// Mitsubishi GX Developer project: 101-Aug09_20121119   PLC: FX1N

PROGRAM MAIN
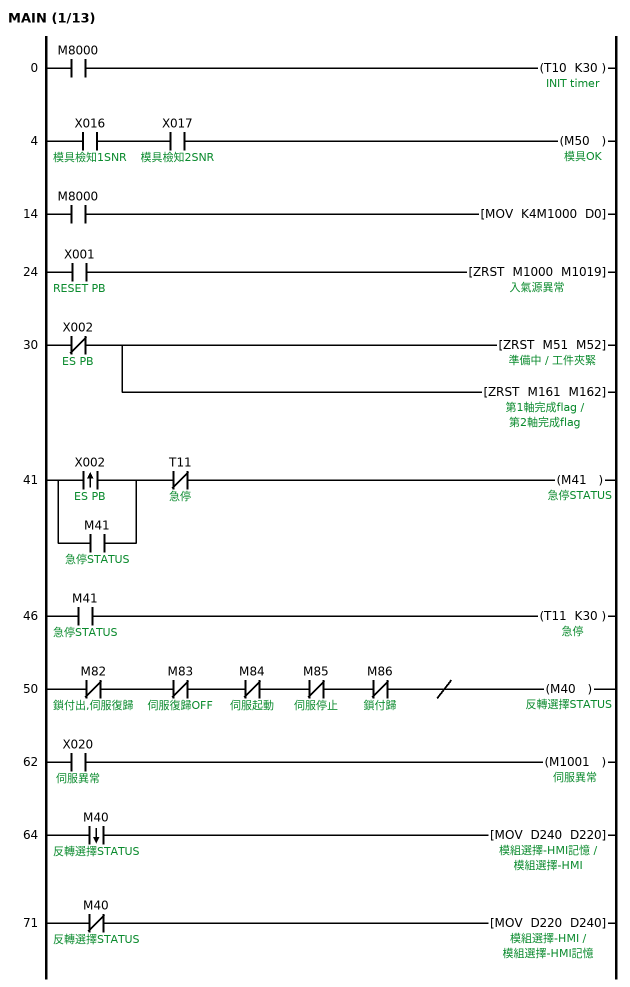
0     LD      M8000
      OUT     T10 K30  ; INIT timer
4     LD      X016  ; 模具檢知1SNR
      AND     X017  ; 模具檢知2SNR
      OUT     M50  ; 模具OK
14    LD      M8000
      MOV     K4M1000 D0  ; 入氣源異常
24    LD      X001  ; RESET PB
      ZRST    M1000 M1019
30    LDI     X002  ; ES PB
      ZRST    M51 M52  ; 準備中 / 工件夾緊
      ZRST    M161 M162  ; 第1軸完成flag / 第2軸完成flag
41    LDP     X002  ; ES PB
      OR      M41  ; 急停STATUS
      ANI     T11  ; 急停
      OUT     M41  ; 急停STATUS
46    LD      M41  ; 急停STATUS
      OUT     T11 K30  ; 急停
50    LDI     M82  ; 鎖付出,伺服復歸
      ANI     M83  ; 伺服復歸OFF
      ANI     M84  ; 伺服起動
      ANI     M85  ; 伺服停止
      ANI     M86  ; 鎖付歸
      INV
      OUT     M40  ; 反轉選擇STATUS
62    LD      X020  ; 伺服異常
      OUT     M1001  ; 伺服異常
64    LDF     M40  ; 反轉選擇STATUS
      MOV     D240 D220  ; 模組選擇-HMI記憶 / 模組選擇-HMI
71    LDI     M40  ; 反轉選擇STATUS
      MOV     D220 D240
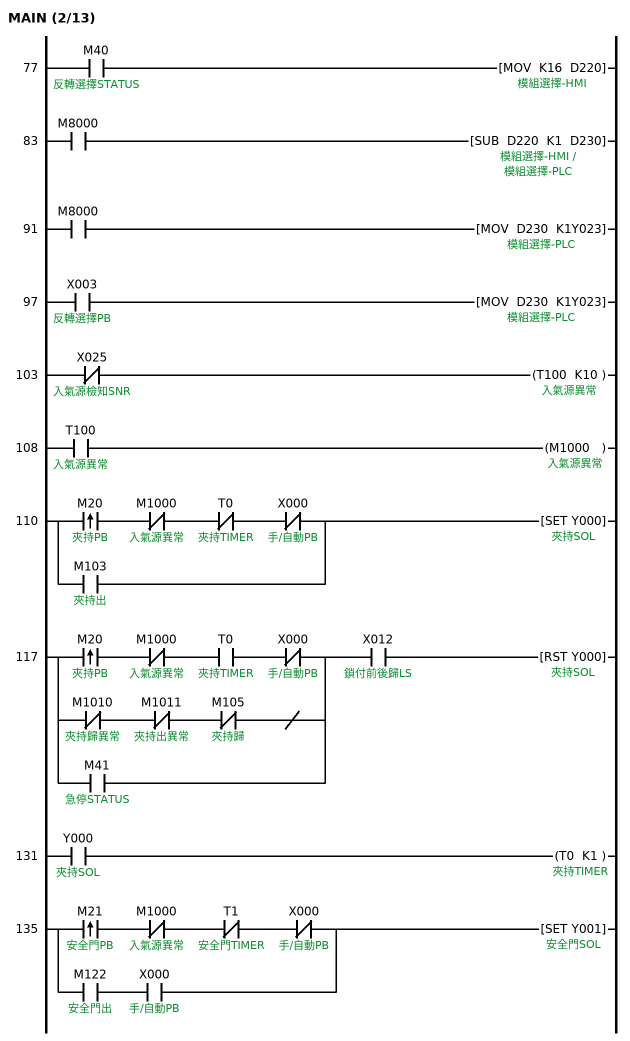
77    LD      M40  ; 反轉選擇STATUS
      MOV     K16 D220
83    LD      M8000
      SUB     D220 K1 D230  ; 模組選擇-PLC
91    LD      M8000
      MOV     D230 K1Y023  ; 工件選擇0
97    LD      X003  ; 反轉選擇PB
      MOV     D230 K1Y023
103   LDI     X025  ; 入氣源檢知SNR
      OUT     T100 K10  ; 入氣源異常
108   LD      T100  ; 入氣源異常
      OUT     M1000  ; 入氣源異常
110   LDP     M20  ; 夾持PB
      ANI     M1000  ; 入氣源異常
      ANI     T0  ; 夾持TIMER
      ANI     X000  ; 手/自動PB
      OR      M103  ; 夾持出
      SET     Y000  ; 夾持SOL
117   LDP     M20  ; 夾持PB
      ANI     M1000  ; 入氣源異常
      AND     T0  ; 夾持TIMER
      ANI     X000  ; 手/自動PB
      LDI     M1010  ; 夾持歸異常
      ANI     M1011  ; 夾持出異常
      ANI     M105  ; 夾持歸
      INV
      ORB
      OR      M41  ; 急停STATUS
      AND     X012  ; 鎖付前後歸LS
      RST     Y000  ; 夾持SOL
131   LD      Y000  ; 夾持SOL
      OUT     T0 K1  ; 夾持TIMER
135   LDP     M21  ; 安全門PB
      ANI     M1000  ; 入氣源異常
      ANI     T1  ; 安全門TIMER
      ANI     X000  ; 手/自動PB
      LD      M122  ; 安全門出
      AND     X000  ; 手/自動PB
      ORB
      SET     Y001  ; 安全門SOL
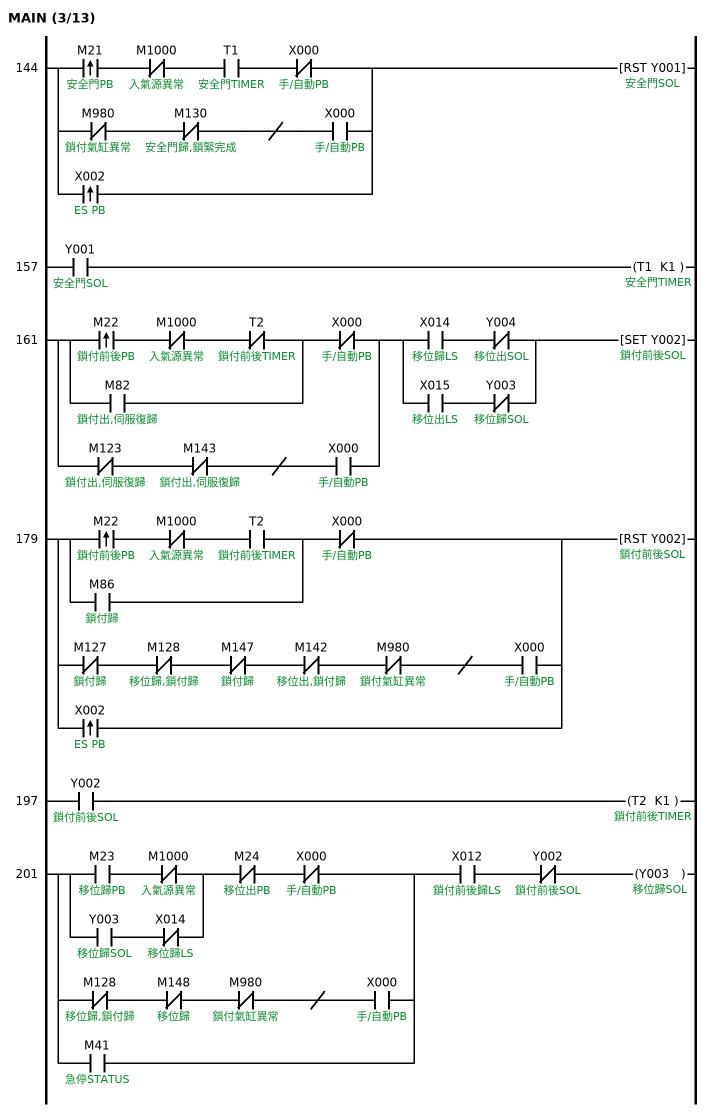
144   LDP     M21  ; 安全門PB
      ANI     M1000  ; 入氣源異常
      AND     T1  ; 安全門TIMER
      ANI     X000  ; 手/自動PB
      LDI     M980  ; 鎖付氣缸異常
      ANI     M130  ; 安全門歸,鎖緊完成
      INV
      AND     X000  ; 手/自動PB
      ORB
      ORP     X002  ; ES PB
      RST     Y001  ; 安全門SOL
157   LD      Y001  ; 安全門SOL
      OUT     T1 K1  ; 安全門TIMER
161   LDP     M22  ; 鎖付前後PB
      ANI     M1000  ; 入氣源異常
      ANI     T2  ; 鎖付前後TIMER
      OR      M82  ; 鎖付出,伺服復歸
      ANI     X000  ; 手/自動PB
      LDI     M123  ; 鎖付出,伺服復歸
      ANI     M143  ; 鎖付出,伺服復歸
      INV
      AND     X000  ; 手/自動PB
      ORB
      LD      X014  ; 移位歸LS
      ANI     Y004  ; 移位出SOL
      LD      X015  ; 移位出LS
      ANI     Y003  ; 移位歸SOL
      ORB
      ANB
      SET     Y002  ; 鎖付前後SOL
179   LDP     M22  ; 鎖付前後PB
      ANI     M1000  ; 入氣源異常
      AND     T2  ; 鎖付前後TIMER
      OR      M86  ; 鎖付歸
      ANI     X000  ; 手/自動PB
      LDI     M127  ; 鎖付歸
      ANI     M128  ; 移位歸,鎖付歸
      ANI     M147  ; 鎖付歸
      ANI     M142  ; 移位出,鎖付歸
      ANI     M980  ; 鎖付氣缸異常
      INV
      AND     X000  ; 手/自動PB
      ORB
      ORP     X002  ; ES PB
      RST     Y002  ; 鎖付前後SOL
197   LD      Y002  ; 鎖付前後SOL
      OUT     T2 K1  ; 鎖付前後TIMER
201   LD      M23  ; 移位歸PB
      ANI     M1000  ; 入氣源異常
      LD      Y003  ; 移位歸SOL
      ANI     X014  ; 移位歸LS
      ORB
      ANI     M24  ; 移位出PB
      ANI     X000  ; 手/自動PB
      LDI     M128  ; 移位歸,鎖付歸
      ANI     M148  ; 移位歸
      ANI     M980  ; 鎖付氣缸異常
      INV
      AND     X000  ; 手/自動PB
      ORB
      OR      M41  ; 急停STATUS
      AND     X012  ; 鎖付前後歸LS
      ANI     Y002  ; 鎖付前後SOL
      OUT     Y003  ; 移位歸SOL
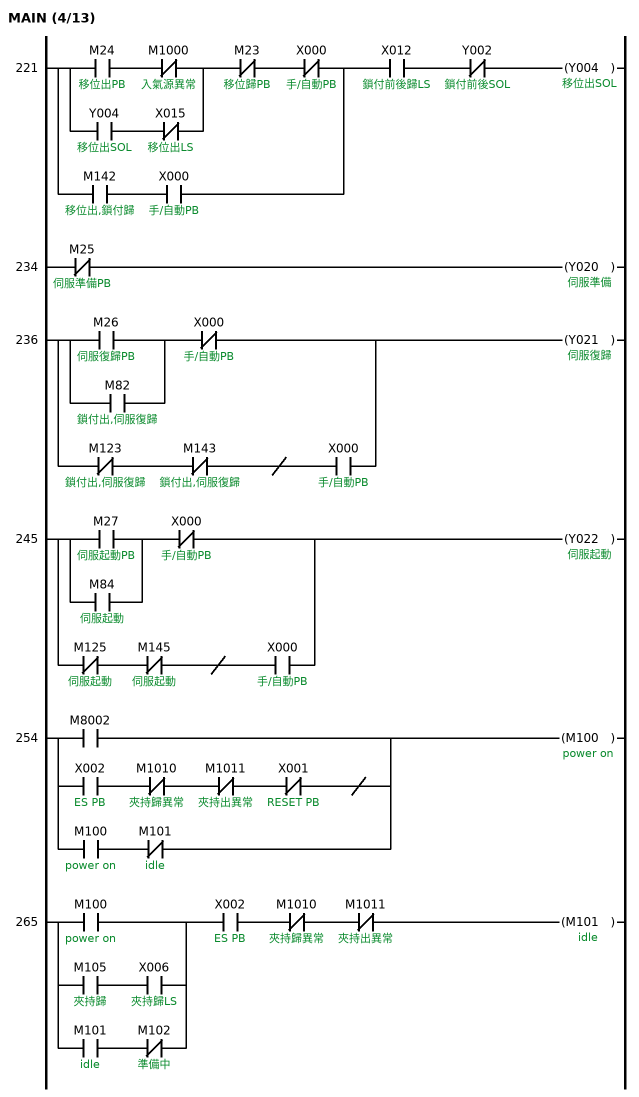
221   LD      M24  ; 移位出PB
      ANI     M1000  ; 入氣源異常
      LD      Y004  ; 移位出SOL
      ANI     X015  ; 移位出LS
      ORB
      ANI     M23  ; 移位歸PB
      ANI     X000  ; 手/自動PB
      LD      M142  ; 移位出,鎖付歸
      AND     X000  ; 手/自動PB
      ORB
      AND     X012  ; 鎖付前後歸LS
      ANI     Y002  ; 鎖付前後SOL
      OUT     Y004  ; 移位出SOL
234   LDI     M25  ; 伺服準備PB
      OUT     Y020  ; 伺服準備
236   LD      M26  ; 伺服復歸PB
      OR      M82  ; 鎖付出,伺服復歸
      ANI     X000  ; 手/自動PB
      LDI     M123  ; 鎖付出,伺服復歸
      ANI     M143  ; 鎖付出,伺服復歸
      INV
      AND     X000  ; 手/自動PB
      ORB
      OUT     Y021  ; 伺服復歸
245   LD      M27  ; 伺服起動PB
      OR      M84  ; 伺服起動
      ANI     X000  ; 手/自動PB
      LDI     M125  ; 伺服起動
      ANI     M145  ; 伺服起動
      INV
      AND     X000  ; 手/自動PB
      ORB
      OUT     Y022  ; 伺服起動
254   LD      M8002
      LD      X002  ; ES PB
      ANI     M1010  ; 夾持歸異常
      ANI     M1011  ; 夾持出異常
      ANI     X001  ; RESET PB
      INV
      ORB
      LD      M100  ; power on
      ANI     M101  ; idle
      ORB
      OUT     M100  ; power on
265   LD      M100  ; power on
      LD      M105  ; 夾持歸
      AND     X006  ; 夾持歸LS
      ORB
      LD      M101  ; idle
      ANI     M102  ; 準備中
      ORB
      AND     X002  ; ES PB
      ANI     M1010  ; 夾持歸異常
      ANI     M1011  ; 夾持出異常
      OUT     M101  ; idle
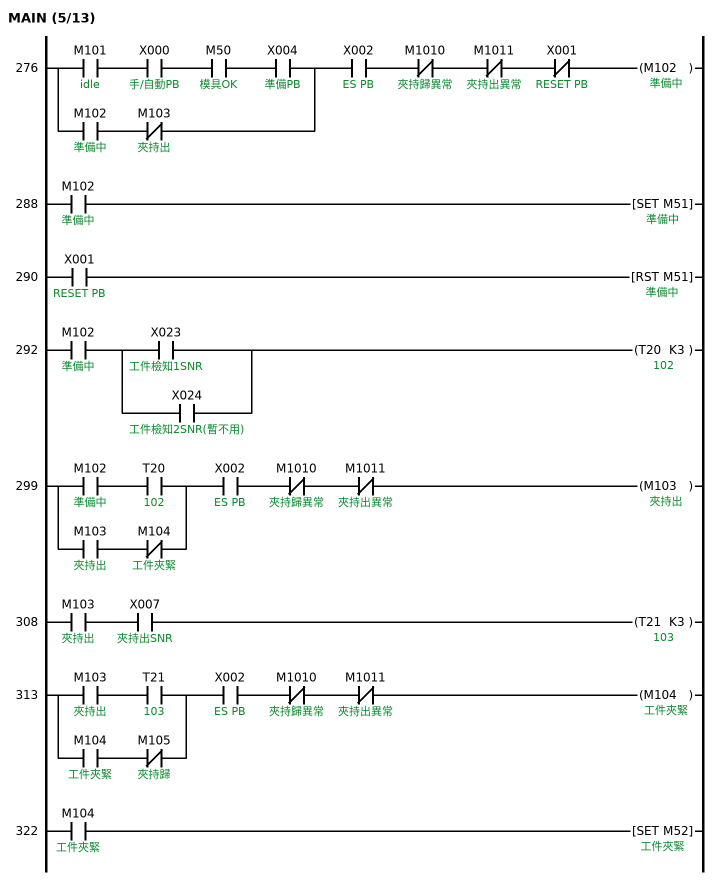
276   LD      M101  ; idle
      AND     X000  ; 手/自動PB
      AND     M50  ; 模具OK
      AND     X004  ; 準備PB
      LD      M102  ; 準備中
      ANI     M103  ; 夾持出
      ORB
      AND     X002  ; ES PB
      ANI     M1010  ; 夾持歸異常
      ANI     M1011  ; 夾持出異常
      ANI     X001  ; RESET PB
      OUT     M102  ; 準備中
288   LD      M102  ; 準備中
      SET     M51  ; 準備中
290   LD      X001  ; RESET PB
      RST     M51  ; 準備中
292   LD      M102  ; 準備中
      LD      X023  ; 工件檢知1SNR
      OR      X024  ; 工件檢知2SNR(暫不用)
      ANB
      OUT     T20 K3  ; 102
299   LD      M102  ; 準備中
      AND     T20  ; 102
      LD      M103  ; 夾持出
      ANI     M104  ; 工件夾緊
      ORB
      AND     X002  ; ES PB
      ANI     M1010  ; 夾持歸異常
      ANI     M1011  ; 夾持出異常
      OUT     M103  ; 夾持出
308   LD      M103  ; 夾持出
      AND     X007  ; 夾持出SNR
      OUT     T21 K3  ; 103
313   LD      M103  ; 夾持出
      AND     T21  ; 103
      LD      M104  ; 工件夾緊
      ANI     M105  ; 夾持歸
      ORB
      AND     X002  ; ES PB
      ANI     M1010  ; 夾持歸異常
      ANI     M1011  ; 夾持出異常
      OUT     M104  ; 工件夾緊
322   LD      M104  ; 工件夾緊
      SET     M52  ; 工件夾緊
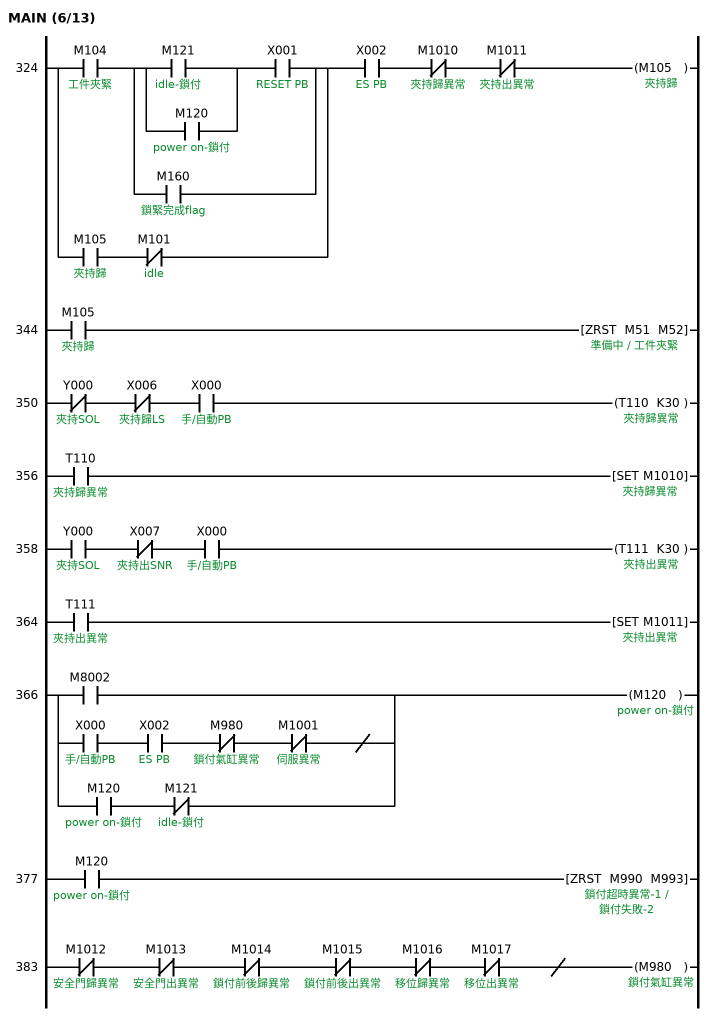
324   LD      M104  ; 工件夾緊
      LD      M121  ; idle-鎖付
      OR      M120  ; power on-鎖付
      AND     X001  ; RESET PB
      OR      M160  ; 鎖緊完成flag
      ANB
      LD      M105  ; 夾持歸
      ANI     M101  ; idle
      ORB
      AND     X002  ; ES PB
      ANI     M1010  ; 夾持歸異常
      ANI     M1011  ; 夾持出異常
      OUT     M105  ; 夾持歸
344   LD      M105  ; 夾持歸
      ZRST    M51 M52
350   LDI     Y000  ; 夾持SOL
      ANI     X006  ; 夾持歸LS
      AND     X000  ; 手/自動PB
      OUT     T110 K30  ; 夾持歸異常
356   LD      T110  ; 夾持歸異常
      SET     M1010  ; 夾持歸異常
358   LD      Y000  ; 夾持SOL
      ANI     X007  ; 夾持出SNR
      AND     X000  ; 手/自動PB
      OUT     T111 K30  ; 夾持出異常
364   LD      T111  ; 夾持出異常
      SET     M1011  ; 夾持出異常
366   LD      M8002
      LD      X000  ; 手/自動PB
      AND     X002  ; ES PB
      ANI     M980  ; 鎖付氣缸異常
      ANI     M1001  ; 伺服異常
      INV
      ORB
      LD      M120  ; power on-鎖付
      ANI     M121  ; idle-鎖付
      ORB
      OUT     M120  ; power on-鎖付
377   LD      M120  ; power on-鎖付
      ZRST    M990 M993  ; 鎖付超時異常-1 / 鎖付失敗-2
383   LDI     M1012  ; 安全門歸異常
      ANI     M1013  ; 安全門出異常
      ANI     M1014  ; 鎖付前後歸異常
      ANI     M1015  ; 鎖付前後出異常
      ANI     M1016  ; 移位歸異常
      ANI     M1017  ; 移位出異常
      INV
      OUT     M980  ; 鎖付氣缸異常
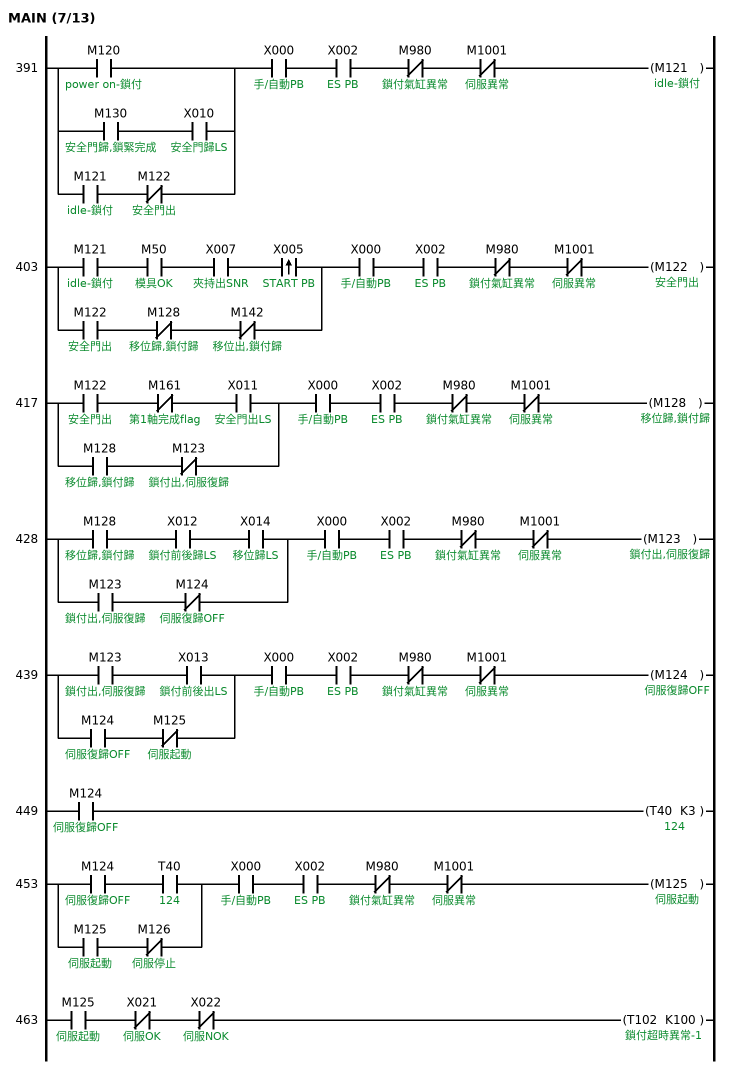
391   LD      M120  ; power on-鎖付
      LD      M130  ; 安全門歸,鎖緊完成
      AND     X010  ; 安全門歸LS
      ORB
      LD      M121  ; idle-鎖付
      ANI     M122  ; 安全門出
      ORB
      AND     X000  ; 手/自動PB
      AND     X002  ; ES PB
      ANI     M980  ; 鎖付氣缸異常
      ANI     M1001  ; 伺服異常
      OUT     M121  ; idle-鎖付
403   LD      M121  ; idle-鎖付
      AND     M50  ; 模具OK
      AND     X007  ; 夾持出SNR
      ANDP    X005  ; START PB
      LD      M122  ; 安全門出
      ANI     M128  ; 移位歸,鎖付歸
      ANI     M142  ; 移位出,鎖付歸
      ORB
      AND     X000  ; 手/自動PB
      AND     X002  ; ES PB
      ANI     M980  ; 鎖付氣缸異常
      ANI     M1001  ; 伺服異常
      OUT     M122  ; 安全門出
417   LD      M122  ; 安全門出
      ANI     M161  ; 第1軸完成flag
      AND     X011  ; 安全門出LS
      LD      M128  ; 移位歸,鎖付歸
      ANI     M123  ; 鎖付出,伺服復歸
      ORB
      AND     X000  ; 手/自動PB
      AND     X002  ; ES PB
      ANI     M980  ; 鎖付氣缸異常
      ANI     M1001  ; 伺服異常
      OUT     M128  ; 移位歸,鎖付歸
428   LD      M128  ; 移位歸,鎖付歸
      AND     X012  ; 鎖付前後歸LS
      AND     X014  ; 移位歸LS
      LD      M123  ; 鎖付出,伺服復歸
      ANI     M124  ; 伺服復歸OFF
      ORB
      AND     X000  ; 手/自動PB
      AND     X002  ; ES PB
      ANI     M980  ; 鎖付氣缸異常
      ANI     M1001  ; 伺服異常
      OUT     M123  ; 鎖付出,伺服復歸
439   LD      M123  ; 鎖付出,伺服復歸
      AND     X013  ; 鎖付前後出LS
      LD      M124  ; 伺服復歸OFF
      ANI     M125  ; 伺服起動
      ORB
      AND     X000  ; 手/自動PB
      AND     X002  ; ES PB
      ANI     M980  ; 鎖付氣缸異常
      ANI     M1001  ; 伺服異常
      OUT     M124  ; 伺服復歸OFF
449   LD      M124  ; 伺服復歸OFF
      OUT     T40 K3  ; 124
453   LD      M124  ; 伺服復歸OFF
      AND     T40  ; 124
      LD      M125  ; 伺服起動
      ANI     M126  ; 伺服停止
      ORB
      AND     X000  ; 手/自動PB
      AND     X002  ; ES PB
      ANI     M980  ; 鎖付氣缸異常
      ANI     M1001  ; 伺服異常
      OUT     M125  ; 伺服起動
463   LD      M125  ; 伺服起動
      ANI     X021  ; 伺服OK
      ANI     X022  ; 伺服NOK
      OUT     T102 K100  ; 鎖付超時異常-1
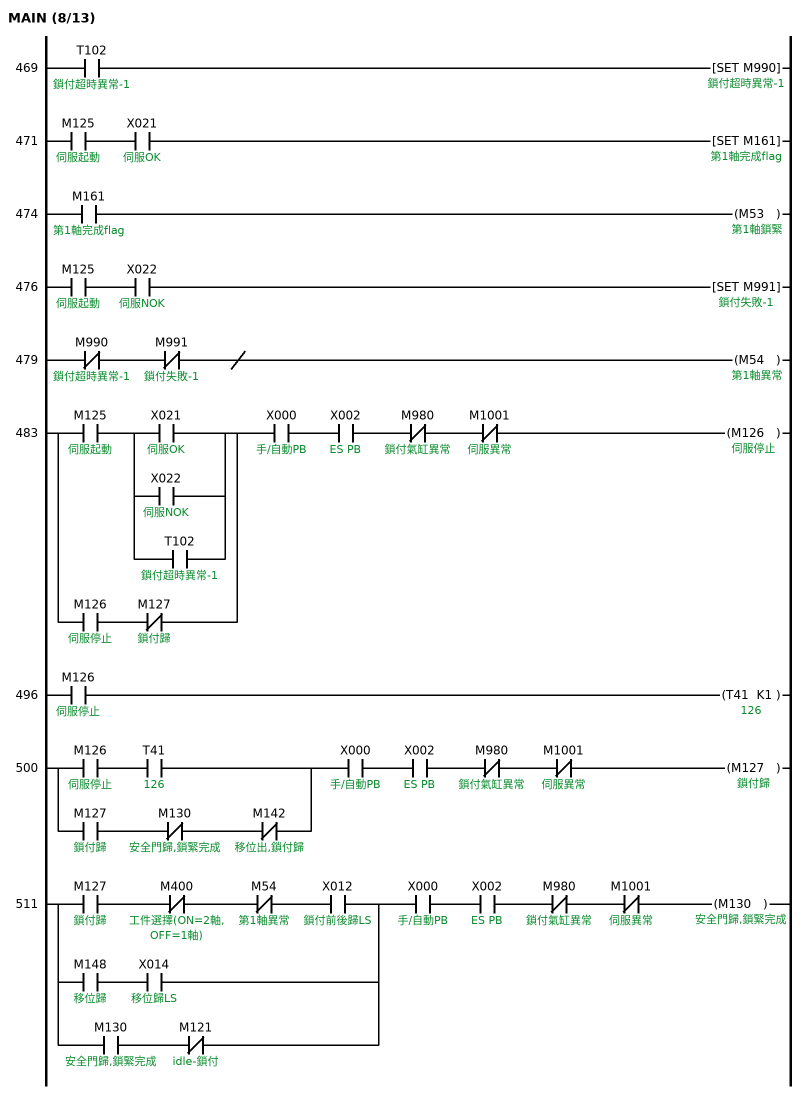
469   LD      T102  ; 鎖付超時異常-1
      SET     M990  ; 鎖付超時異常-1
471   LD      M125  ; 伺服起動
      AND     X021  ; 伺服OK
      SET     M161  ; 第1軸完成flag
474   LD      M161  ; 第1軸完成flag
      OUT     M53  ; 第1軸鎖緊
476   LD      M125  ; 伺服起動
      AND     X022  ; 伺服NOK
      SET     M991  ; 鎖付失敗-1
479   LDI     M990  ; 鎖付超時異常-1
      ANI     M991  ; 鎖付失敗-1
      INV
      OUT     M54  ; 第1軸異常
483   LD      M125  ; 伺服起動
      LD      X021  ; 伺服OK
      OR      X022  ; 伺服NOK
      OR      T102  ; 鎖付超時異常-1
      ANB
      LD      M126  ; 伺服停止
      ANI     M127  ; 鎖付歸
      ORB
      AND     X000  ; 手/自動PB
      AND     X002  ; ES PB
      ANI     M980  ; 鎖付氣缸異常
      ANI     M1001  ; 伺服異常
      OUT     M126  ; 伺服停止
496   LD      M126  ; 伺服停止
      OUT     T41 K1  ; 126
500   LD      M126  ; 伺服停止
      AND     T41  ; 126
      LD      M127  ; 鎖付歸
      ANI     M130  ; 安全門歸,鎖緊完成
      ANI     M142  ; 移位出,鎖付歸
      ORB
      AND     X000  ; 手/自動PB
      AND     X002  ; ES PB
      ANI     M980  ; 鎖付氣缸異常
      ANI     M1001  ; 伺服異常
      OUT     M127  ; 鎖付歸
511   LD      M127  ; 鎖付歸
      ANI     M400  ; 工件選擇(ON=2軸,OFF=1軸)
      ANI     M54  ; 第1軸異常
      AND     X012  ; 鎖付前後歸LS
      LD      M148  ; 移位歸
      AND     X014  ; 移位歸LS
      ORB
      LD      M130  ; 安全門歸,鎖緊完成
      ANI     M121  ; idle-鎖付
      ORB
      AND     X000  ; 手/自動PB
      AND     X002  ; ES PB
      ANI     M980  ; 鎖付氣缸異常
      ANI     M1001  ; 伺服異常
      OUT     M130  ; 安全門歸,鎖緊完成
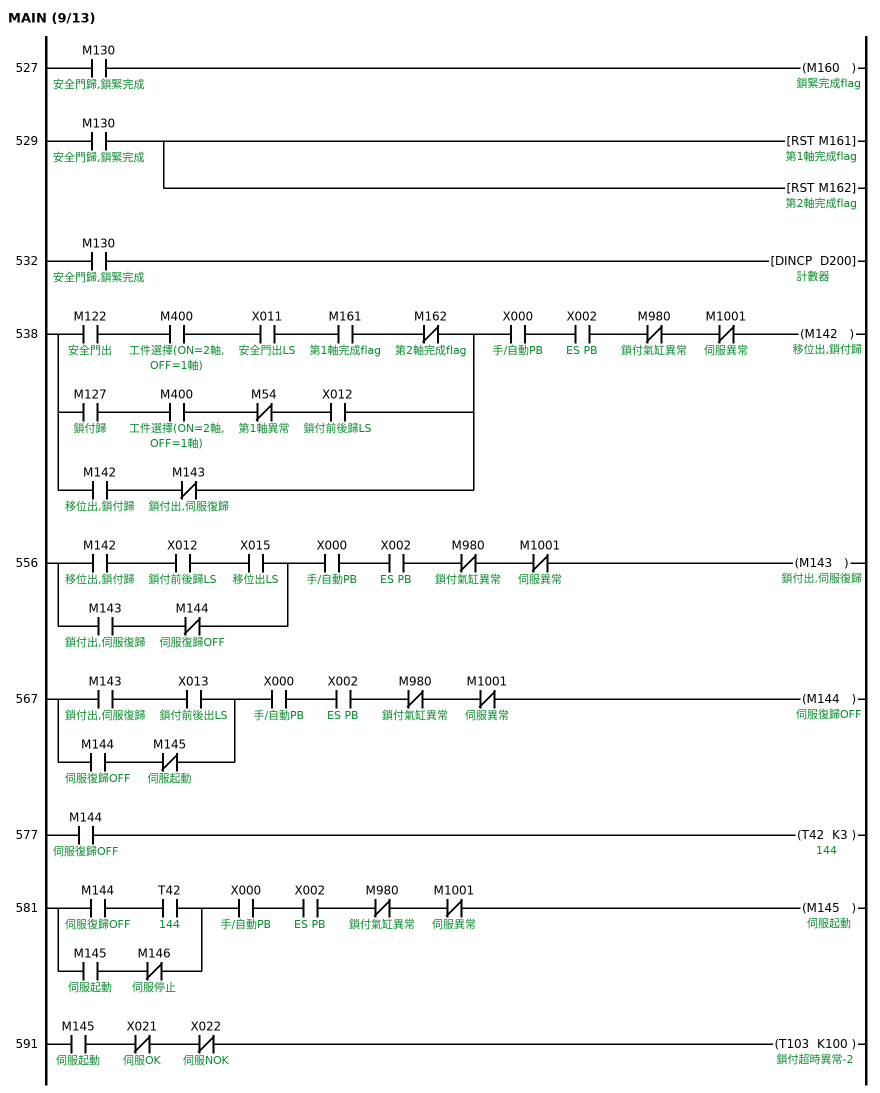
527   LD      M130  ; 安全門歸,鎖緊完成
      OUT     M160  ; 鎖緊完成flag
529   LD      M130  ; 安全門歸,鎖緊完成
      RST     M161  ; 第1軸完成flag
      RST     M162  ; 第2軸完成flag
532   LD      M130  ; 安全門歸,鎖緊完成
      DINCP   D200  ; 計數器
538   LD      M122  ; 安全門出
      AND     M400  ; 工件選擇(ON=2軸,OFF=1軸)
      AND     X011  ; 安全門出LS
      AND     M161  ; 第1軸完成flag
      ANI     M162  ; 第2軸完成flag
      LD      M127  ; 鎖付歸
      AND     M400  ; 工件選擇(ON=2軸,OFF=1軸)
      ANI     M54  ; 第1軸異常
      AND     X012  ; 鎖付前後歸LS
      ORB
      LD      M142  ; 移位出,鎖付歸
      ANI     M143  ; 鎖付出,伺服復歸
      ORB
      AND     X000  ; 手/自動PB
      AND     X002  ; ES PB
      ANI     M980  ; 鎖付氣缸異常
      ANI     M1001  ; 伺服異常
      OUT     M142  ; 移位出,鎖付歸
556   LD      M142  ; 移位出,鎖付歸
      AND     X012  ; 鎖付前後歸LS
      AND     X015  ; 移位出LS
      LD      M143  ; 鎖付出,伺服復歸
      ANI     M144  ; 伺服復歸OFF
      ORB
      AND     X000  ; 手/自動PB
      AND     X002  ; ES PB
      ANI     M980  ; 鎖付氣缸異常
      ANI     M1001  ; 伺服異常
      OUT     M143  ; 鎖付出,伺服復歸
567   LD      M143  ; 鎖付出,伺服復歸
      AND     X013  ; 鎖付前後出LS
      LD      M144  ; 伺服復歸OFF
      ANI     M145  ; 伺服起動
      ORB
      AND     X000  ; 手/自動PB
      AND     X002  ; ES PB
      ANI     M980  ; 鎖付氣缸異常
      ANI     M1001  ; 伺服異常
      OUT     M144  ; 伺服復歸OFF
577   LD      M144  ; 伺服復歸OFF
      OUT     T42 K3  ; 144
581   LD      M144  ; 伺服復歸OFF
      AND     T42  ; 144
      LD      M145  ; 伺服起動
      ANI     M146  ; 伺服停止
      ORB
      AND     X000  ; 手/自動PB
      AND     X002  ; ES PB
      ANI     M980  ; 鎖付氣缸異常
      ANI     M1001  ; 伺服異常
      OUT     M145  ; 伺服起動
591   LD      M145  ; 伺服起動
      ANI     X021  ; 伺服OK
      ANI     X022  ; 伺服NOK
      OUT     T103 K100  ; 鎖付超時異常-2
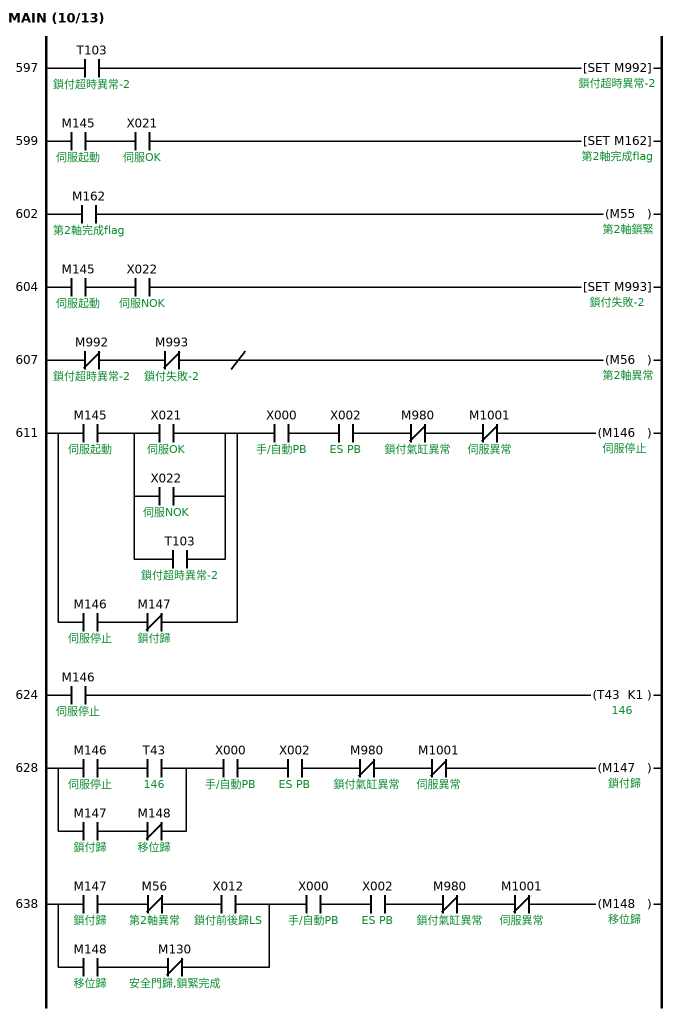
597   LD      T103  ; 鎖付超時異常-2
      SET     M992  ; 鎖付超時異常-2
599   LD      M145  ; 伺服起動
      AND     X021  ; 伺服OK
      SET     M162  ; 第2軸完成flag
602   LD      M162  ; 第2軸完成flag
      OUT     M55  ; 第2軸鎖緊
604   LD      M145  ; 伺服起動
      AND     X022  ; 伺服NOK
      SET     M993  ; 鎖付失敗-2
607   LDI     M992  ; 鎖付超時異常-2
      ANI     M993  ; 鎖付失敗-2
      INV
      OUT     M56  ; 第2軸異常
611   LD      M145  ; 伺服起動
      LD      X021  ; 伺服OK
      OR      X022  ; 伺服NOK
      OR      T103  ; 鎖付超時異常-2
      ANB
      LD      M146  ; 伺服停止
      ANI     M147  ; 鎖付歸
      ORB
      AND     X000  ; 手/自動PB
      AND     X002  ; ES PB
      ANI     M980  ; 鎖付氣缸異常
      ANI     M1001  ; 伺服異常
      OUT     M146  ; 伺服停止
624   LD      M146  ; 伺服停止
      OUT     T43 K1  ; 146
628   LD      M146  ; 伺服停止
      AND     T43  ; 146
      LD      M147  ; 鎖付歸
      ANI     M148  ; 移位歸
      ORB
      AND     X000  ; 手/自動PB
      AND     X002  ; ES PB
      ANI     M980  ; 鎖付氣缸異常
      ANI     M1001  ; 伺服異常
      OUT     M147  ; 鎖付歸
638   LD      M147  ; 鎖付歸
      ANI     M56  ; 第2軸異常
      AND     X012  ; 鎖付前後歸LS
      LD      M148  ; 移位歸
      ANI     M130  ; 安全門歸,鎖緊完成
      ORB
      AND     X000  ; 手/自動PB
      AND     X002  ; ES PB
      ANI     M980  ; 鎖付氣缸異常
      ANI     M1001  ; 伺服異常
      OUT     M148  ; 移位歸
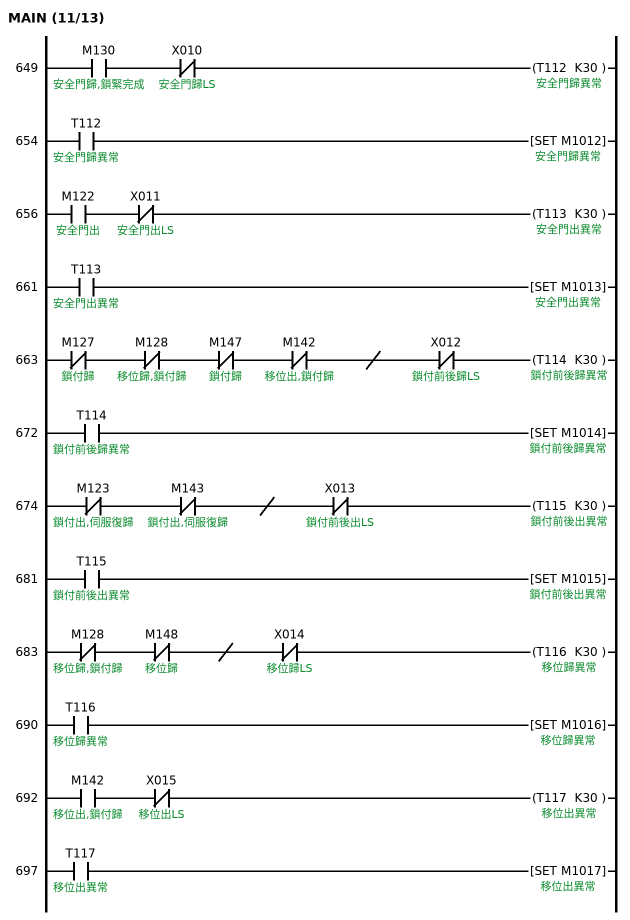
649   LD      M130  ; 安全門歸,鎖緊完成
      ANI     X010  ; 安全門歸LS
      OUT     T112 K30  ; 安全門歸異常
654   LD      T112  ; 安全門歸異常
      SET     M1012  ; 安全門歸異常
656   LD      M122  ; 安全門出
      ANI     X011  ; 安全門出LS
      OUT     T113 K30  ; 安全門出異常
661   LD      T113  ; 安全門出異常
      SET     M1013  ; 安全門出異常
663   LDI     M127  ; 鎖付歸
      ANI     M128  ; 移位歸,鎖付歸
      ANI     M147  ; 鎖付歸
      ANI     M142  ; 移位出,鎖付歸
      INV
      ANI     X012  ; 鎖付前後歸LS
      OUT     T114 K30  ; 鎖付前後歸異常
672   LD      T114  ; 鎖付前後歸異常
      SET     M1014  ; 鎖付前後歸異常
674   LDI     M123  ; 鎖付出,伺服復歸
      ANI     M143  ; 鎖付出,伺服復歸
      INV
      ANI     X013  ; 鎖付前後出LS
      OUT     T115 K30  ; 鎖付前後出異常
681   LD      T115  ; 鎖付前後出異常
      SET     M1015  ; 鎖付前後出異常
683   LDI     M128  ; 移位歸,鎖付歸
      ANI     M148  ; 移位歸
      INV
      ANI     X014  ; 移位歸LS
      OUT     T116 K30  ; 移位歸異常
690   LD      T116  ; 移位歸異常
      SET     M1016  ; 移位歸異常
692   LD      M142  ; 移位出,鎖付歸
      ANI     X015  ; 移位出LS
      OUT     T117 K30  ; 移位出異常
697   LD      T117  ; 移位出異常
      SET     M1017  ; 移位出異常
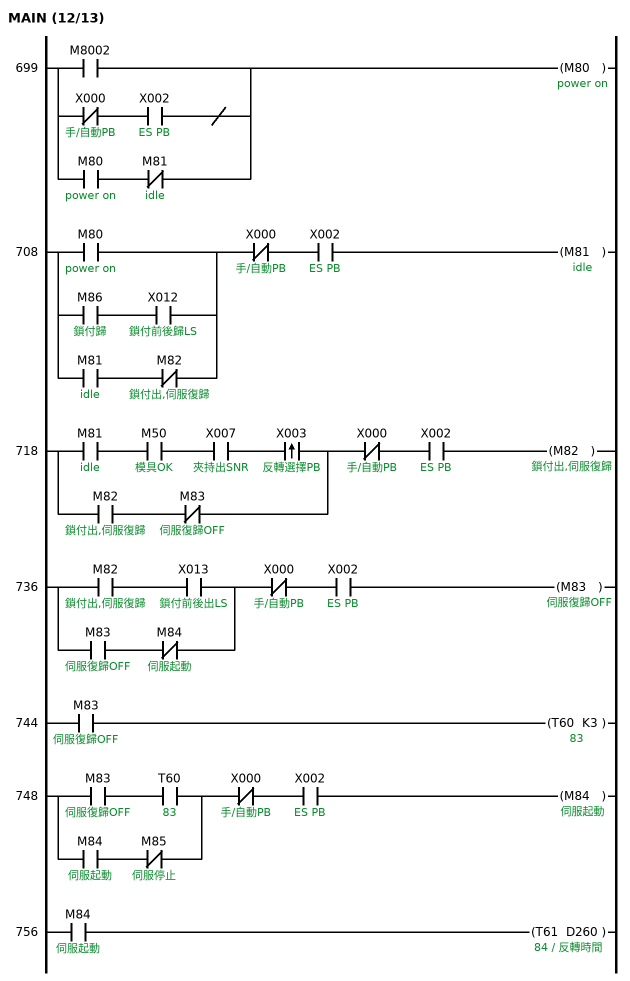
699   LD      M8002
      LDI     X000  ; 手/自動PB
      AND     X002  ; ES PB
      INV
      ORB
      LD      M80  ; power on
      ANI     M81  ; idle
      ORB
      OUT     M80  ; power on
708   LD      M80  ; power on
      LD      M86  ; 鎖付歸
      AND     X012  ; 鎖付前後歸LS
      ORB
      LD      M81  ; idle
      ANI     M82  ; 鎖付出,伺服復歸
      ORB
      ANI     X000  ; 手/自動PB
      AND     X002  ; ES PB
      OUT     M81  ; idle
718   LD      M81  ; idle
      AND     M50  ; 模具OK
      AND     X007  ; 夾持出SNR
      ANDP    X003  ; 反轉選擇PB
      LD      M82  ; 鎖付出,伺服復歸
      ANI     M83  ; 伺服復歸OFF
      ORB
      ANI     X000  ; 手/自動PB
      AND     X002  ; ES PB
      OUT     M82  ; 鎖付出,伺服復歸
736   LD      M82  ; 鎖付出,伺服復歸
      AND     X013  ; 鎖付前後出LS
      LD      M83  ; 伺服復歸OFF
      ANI     M84  ; 伺服起動
      ORB
      ANI     X000  ; 手/自動PB
      AND     X002  ; ES PB
      OUT     M83  ; 伺服復歸OFF
744   LD      M83  ; 伺服復歸OFF
      OUT     T60 K3  ; 83
748   LD      M83  ; 伺服復歸OFF
      AND     T60  ; 83
      LD      M84  ; 伺服起動
      ANI     M85  ; 伺服停止
      ORB
      ANI     X000  ; 手/自動PB
      AND     X002  ; ES PB
      OUT     M84  ; 伺服起動
756   LD      M84  ; 伺服起動
      OUT     T61 D260  ; 84 / 反轉時間
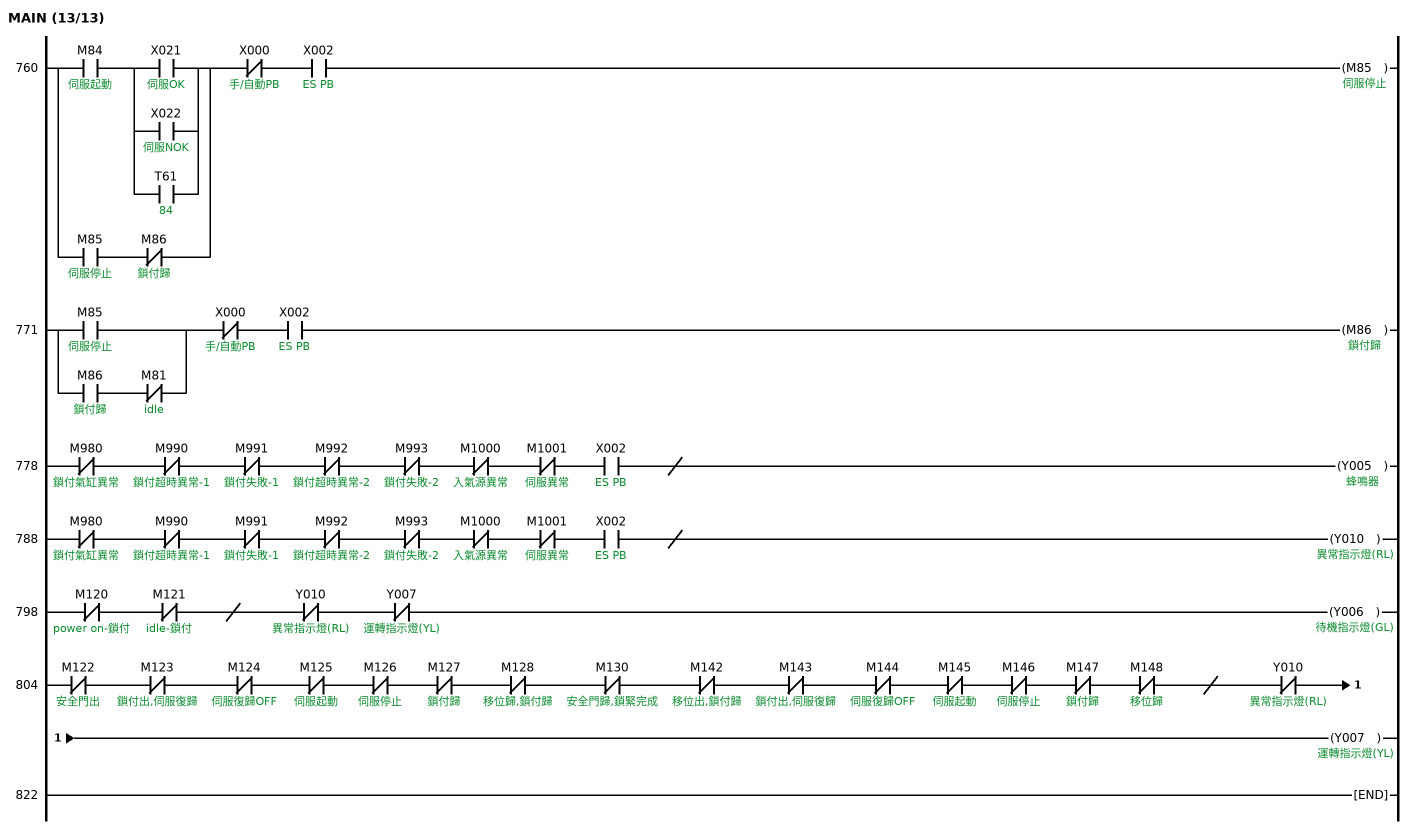
760   LD      M84  ; 伺服起動
      LD      X021  ; 伺服OK
      OR      X022  ; 伺服NOK
      OR      T61  ; 84
      ANB
      LD      M85  ; 伺服停止
      ANI     M86  ; 鎖付歸
      ORB
      ANI     X000  ; 手/自動PB
      AND     X002  ; ES PB
      OUT     M85  ; 伺服停止
771   LD      M85  ; 伺服停止
      LD      M86  ; 鎖付歸
      ANI     M81  ; idle
      ORB
      ANI     X000  ; 手/自動PB
      AND     X002  ; ES PB
      OUT     M86  ; 鎖付歸
778   LDI     M980  ; 鎖付氣缸異常
      ANI     M990  ; 鎖付超時異常-1
      ANI     M991  ; 鎖付失敗-1
      ANI     M992  ; 鎖付超時異常-2
      ANI     M993  ; 鎖付失敗-2
      ANI     M1000  ; 入氣源異常
      ANI     M1001  ; 伺服異常
      AND     X002  ; ES PB
      INV
      OUT     Y005  ; 蜂鳴器
788   LDI     M980  ; 鎖付氣缸異常
      ANI     M990  ; 鎖付超時異常-1
      ANI     M991  ; 鎖付失敗-1
      ANI     M992  ; 鎖付超時異常-2
      ANI     M993  ; 鎖付失敗-2
      ANI     M1000  ; 入氣源異常
      ANI     M1001  ; 伺服異常
      AND     X002  ; ES PB
      INV
      OUT     Y010  ; 異常指示燈(RL)
798   LDI     M120  ; power on-鎖付
      ANI     M121  ; idle-鎖付
      INV
      ANI     Y010  ; 異常指示燈(RL)
      ANI     Y007  ; 運轉指示燈(YL)
      OUT     Y006  ; 待機指示燈(GL)
804   LDI     M122  ; 安全門出
      ANI     M123  ; 鎖付出,伺服復歸
      ANI     M124  ; 伺服復歸OFF
      ANI     M125  ; 伺服起動
      ANI     M126  ; 伺服停止
      ANI     M127  ; 鎖付歸
      ANI     M128  ; 移位歸,鎖付歸
      ANI     M130  ; 安全門歸,鎖緊完成
      ANI     M142  ; 移位出,鎖付歸
      ANI     M143  ; 鎖付出,伺服復歸
      ANI     M144  ; 伺服復歸OFF
      ANI     M145  ; 伺服起動
      ANI     M146  ; 伺服停止
      ANI     M147  ; 鎖付歸
      ANI     M148  ; 移位歸
      INV
      ANI     Y010  ; 異常指示燈(RL)
      OUT     Y007  ; 運轉指示燈(YL)
822   END
END_PROGRAM

// device comments not shown above
Y024  ; 工件選擇1
Y025  ; 工件選擇2
Y026  ; 工件選擇3
Y027  ; 備用
D201  ; 計數器
T3  ; 反轉選擇TIMER
T101  ; 伺服異常
